// TIA Portal V19 export
ORGANIZATION_BLOCK "Main"   // OB1, LAD, ProgramCycle
TITLE = "Main Program Sweep (Cycle)"
{ S7_Optimized_Access := 'TRUE' }
// stored: SetENOAutomatically false
   VAR_INPUT
      Initial_Call : Bool;   // Initial call of this OB
      Remanence : Bool;   // =True, if remanent data are available
   END_VAR
   VAR_TEMP   // added for the SCL form of the ladder/FBD networks
      _w1 : Bool;
      _w2 : Bool;
      _w3 : Bool;
      _w4 : Bool;
   END_VAR
BEGIN

REGION Network 1
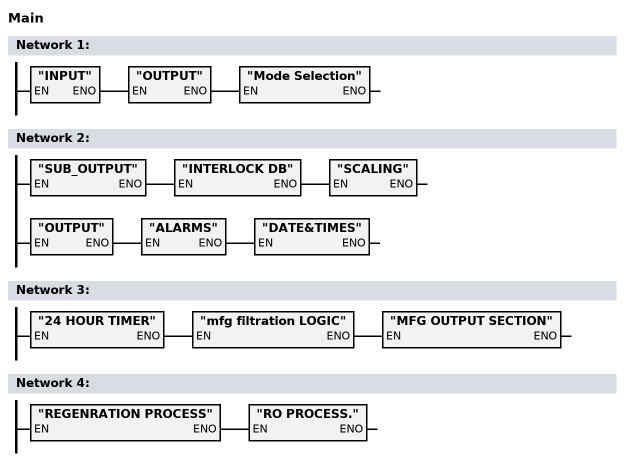
   RUNG wire#powerrail
      "INPUT"()
      "OUTPUT"()
      "Mode Selection"()
   END_RUNG
   // the same network as SCL:
   "INPUT"(ENO => #_w1);
   "OUTPUT"(EN := #_w1, ENO => #_w2);
   IF #_w2 THEN "Mode Selection"(); END_IF;
END_REGION

REGION Network 2
   RUNG wire#powerrail
      "SUB_OUTPUT"()
      "INTERLOCK DB"()
      "SCALING"()
   END_RUNG
   RUNG wire#powerrail
      "OUTPUT"()
      "ALARMS"()
      "DATE&TIMES"()
   END_RUNG
   // the same network as SCL:
   "SUB_OUTPUT"(ENO => #_w1);
   "INTERLOCK DB"(EN := #_w1, ENO => #_w2);
   IF #_w2 THEN "SCALING"(); END_IF;
   "OUTPUT"(ENO => #_w3);
   "ALARMS"(EN := #_w3, ENO => #_w4);
   IF #_w4 THEN "DATE&TIMES"(); END_IF;
END_REGION

REGION Network 3
   RUNG wire#powerrail
      "24 HOUR TIMER"()
      "mfg filtration LOGIC"()
      "MFG OUTPUT SECTION"()
   END_RUNG
   // the same network as SCL:
   "24 HOUR TIMER"(ENO => #_w1);
   "mfg filtration LOGIC"(EN := #_w1, ENO => #_w2);
   IF #_w2 THEN "MFG OUTPUT SECTION"(); END_IF;
END_REGION

REGION Network 4
   RUNG wire#powerrail
      "REGENRATION PROCESS"()
      "RO PROCESS."()
   END_RUNG
   // the same network as SCL:
   "REGENRATION PROCESS"(ENO => #_w1);
   IF #_w1 THEN "RO PROCESS."(); END_IF;
END_REGION
END_ORGANIZATION_BLOCK
